// TIA Portal V20 export
DATA_BLOCK "Config"   // DB7
{ DB_Accessible_From_OPC_UA := 'FALSE' }
AUTHOR : ERsystem_FA2_DH. Kim
// stored: DBAccessibleFromOPCUA false, DBAccessibleFromWebserver false, MemoryReserve 100, Namespace Unit1
   VAR
      unit { S7_SetPoint := 'True'} : "LAF_typeUnitConfiguration";   // Configuration of Unit Parameters
      stateMachine { S7_SetPoint := 'True'} : "LUC_typeStateMachineConfiguration";
      signalStack { S7_SetPoint := 'True'} : "LUC_typeSignalStackConfiguration";
      remoteCtrlOpcUa { S7_SetPoint := 'True'} : "LUC_typeRemoteCtrlConfiguration";
      stateModeManager { ExternalAccessible := 'False'; ExternalVisible := 'False'; ExternalWritable := 'False'} : "LPMLV2022_typeConfiguration";   // Do not change. Can be configured through stateMachineConfiguration
      cmPowerMeter_PAC3220 { S7_SetPoint := 'True'} : "LER_typePAC3220Configuration";
      cmHandyQRreadDM8700 { S7_SetPoint := 'True'} : "LER_typeDM8700Configuration";
      cmFFU_LIU117 { S7_SetPoint := 'True'} : "LER_typeLIU117Configuration";
      sleep { S7_SetPoint := 'True'} : "LER_typeSleepModeParameter";
      BA010 : "LER_typeCommunicationConfiguration";
      BA015 : "LER_typeCommunicationConfiguration";
      BA060 : "LER_typeCommunicationConfiguration";
      BA030 : "LER_typeCommunicationConfiguration";
   END_VAR
BEGIN
   unit.referenceDesignator.parent := WSTRING#'';
   unit.referenceDesignator.relative := WSTRING#'STACK#1';
   unit.referenceDesignator.combined := WSTRING#'STACK#1';
   stateMachine.enableModes.production := TRUE;
   stateMachine.enableModes.maintenance := TRUE;
   stateMachine.enableModes.manual := TRUE;
   stateMachine.enableModes.userMode01 := TRUE;   // Enable unit mode NoMode
   stateMachine.enableModes.userMode02 := TRUE;   // Enable unit mode Sleep
   stateMachine.enableModes.userMode03 := TRUE;   // Enable unit mode DeepSleep
   stateMachine.enableModes.userMode04 := FALSE;
   stateMachine.enableModes.userMode05 := FALSE;
   stateMachine.enableModes.userMode06 := FALSE;
   stateMachine.enableModes.userMode07 := FALSE;
   stateMachine.enableModes.userMode08 := FALSE;
   stateMachine.enableModes.userMode09 := FALSE;
   stateMachine.enableModes.userMode10 := FALSE;
   stateMachine.enableModes.userMode11 := FALSE;
   stateMachine.enableModes.userMode12 := FALSE;
   stateMachine.enableModes.userMode13 := FALSE;
   stateMachine.enableStates[0..16].clearing := TRUE;
   stateMachine.enableStates[0..2].starting := TRUE;
   stateMachine.enableStates[3].starting := FALSE;
   stateMachine.enableStates[4..16].starting := TRUE;
   stateMachine.enableStates[0..1].suspended := TRUE;
   stateMachine.enableStates[2..3].suspended := FALSE;
   stateMachine.enableStates[4..16].suspended := TRUE;
   stateMachine.enableStates[0..16].stopping := TRUE;
   stateMachine.enableStates[0..16].aborting := TRUE;
   stateMachine.enableStates[0..2].holding := TRUE;
   stateMachine.enableStates[3].holding := FALSE;
   stateMachine.enableStates[4..16].holding := TRUE;
   stateMachine.enableStates[0..2].held := TRUE;
   stateMachine.enableStates[3].held := FALSE;
   stateMachine.enableStates[4..16].held := TRUE;
   stateMachine.enableStates[0..2].unholding := TRUE;
   stateMachine.enableStates[3].unholding := FALSE;
   stateMachine.enableStates[4..16].unholding := TRUE;
   stateMachine.enableStates[0..1].suspending := TRUE;
   stateMachine.enableStates[2..3].suspending := FALSE;
   stateMachine.enableStates[4..16].suspending := TRUE;
   stateMachine.enableStates[0..1].unsuspending := TRUE;
   stateMachine.enableStates[2..3].unsuspending := FALSE;
   stateMachine.enableStates[4..16].unsuspending := TRUE;
   stateMachine.enableStates[0..16].resetting := TRUE;
   stateMachine.enableStates[0..1].completing := TRUE;
   stateMachine.enableStates[2..3].completing := FALSE;
   stateMachine.enableStates[4..16].completing := TRUE;
   stateMachine.enableStates[0..1].completed := TRUE;
   stateMachine.enableStates[2..3].completed := FALSE;
   stateMachine.enableStates[4..16].completed := TRUE;
   stateMachine.enableModeTransitions[0..16].clearing := FALSE;
   stateMachine.enableModeTransitions[0..16].stopped := TRUE;
   stateMachine.enableModeTransitions[0..16].starting := FALSE;
   stateMachine.enableModeTransitions[0..16].idle := TRUE;
   stateMachine.enableModeTransitions[0..16].suspended := FALSE;
   stateMachine.enableModeTransitions[0..16].execute := FALSE;
   stateMachine.enableModeTransitions[0..16].stopping := FALSE;
   stateMachine.enableModeTransitions[0..16].aborting := FALSE;
   stateMachine.enableModeTransitions[0..16].aborted := TRUE;
   stateMachine.enableModeTransitions[0..16].holding := FALSE;
   stateMachine.enableModeTransitions[0..16].held := FALSE;
   stateMachine.enableModeTransitions[0..16].unholding := FALSE;
   stateMachine.enableModeTransitions[0..16].suspending := FALSE;
   stateMachine.enableModeTransitions[0..16].unsuspending := FALSE;
   stateMachine.enableModeTransitions[0..16].resetting := FALSE;
   stateMachine.enableModeTransitions[0..16].completing := FALSE;
   stateMachine.enableModeTransitions[0..16].completed := FALSE;
   stateMachine.enableHoldCommand.idle := FALSE;
   stateMachine.enableHoldCommand.starting := FALSE;
   stateMachine.enableHoldCommand.suspended := FALSE;
   stateMachine.enableHoldCommand.execute := TRUE;
   stateMachine.enableHoldCommand.unholding := FALSE;
   stateMachine.enableHoldCommand.suspending := FALSE;
   stateMachine.enableHoldCommand.unsuspending := FALSE;
   stateMachine.enableHoldCommand.completing := FALSE;
   stateMachine.enableHoldCommand.completed := FALSE;
   stateMachine.enableCompleteCommand.suspended := TRUE;
   stateMachine.enableCompleteCommand.execute := TRUE;
   stateMachine.enableCompleteCommand.held := TRUE;
   signalStack.undefined.static.red := FALSE;
   signalStack.undefined.static.yellow := FALSE;
   signalStack.undefined.static.blue := FALSE;
   signalStack.undefined.static.green := FALSE;
   signalStack.undefined.static.horn := FALSE;
   signalStack.undefined.static.white := FALSE;
   signalStack.undefined.static.user1 := FALSE;
   signalStack.undefined.static.user2 := FALSE;
   signalStack.undefined.flashing.red := TRUE;
   signalStack.undefined.flashing.yellow := FALSE;
   signalStack.undefined.flashing.blue := FALSE;
   signalStack.undefined.flashing.green := FALSE;
   signalStack.undefined.flashing.horn := FALSE;
   signalStack.undefined.flashing.white := FALSE;
   signalStack.undefined.flashing.user1 := FALSE;
   signalStack.undefined.flashing.user2 := FALSE;
   signalStack.clearing.static.red := FALSE;
   signalStack.clearing.static.yellow := FALSE;
   signalStack.clearing.static.blue := FALSE;
   signalStack.clearing.static.green := FALSE;
   signalStack.clearing.static.horn := FALSE;
   signalStack.clearing.static.white := FALSE;
   signalStack.clearing.static.user1 := FALSE;
   signalStack.clearing.static.user2 := FALSE;
   signalStack.clearing.flashing.red := TRUE;
   signalStack.clearing.flashing.yellow := FALSE;
   signalStack.clearing.flashing.blue := FALSE;
   signalStack.clearing.flashing.green := FALSE;
   signalStack.clearing.flashing.horn := FALSE;
   signalStack.clearing.flashing.white := FALSE;
   signalStack.clearing.flashing.user1 := FALSE;
   signalStack.clearing.flashing.user2 := FALSE;
   signalStack.stopped.static.red := TRUE;
   signalStack.stopped.static.yellow := FALSE;
   signalStack.stopped.static.blue := FALSE;
   signalStack.stopped.static.green := FALSE;
   signalStack.stopped.static.horn := FALSE;
   signalStack.stopped.static.white := FALSE;
   signalStack.stopped.static.user1 := FALSE;
   signalStack.stopped.static.user2 := FALSE;
   signalStack.stopped.flashing.red := FALSE;
   signalStack.stopped.flashing.yellow := FALSE;
   signalStack.stopped.flashing.blue := FALSE;
   signalStack.stopped.flashing.green := FALSE;
   signalStack.stopped.flashing.horn := FALSE;
   signalStack.stopped.flashing.white := FALSE;
   signalStack.stopped.flashing.user1 := FALSE;
   signalStack.stopped.flashing.user2 := FALSE;
   signalStack.starting.static.red := FALSE;
   signalStack.starting.static.yellow := FALSE;
   signalStack.starting.static.blue := FALSE;
   signalStack.starting.static.green := TRUE;
   signalStack.starting.static.horn := FALSE;
   signalStack.starting.static.white := FALSE;
   signalStack.starting.static.user1 := FALSE;
   signalStack.starting.static.user2 := FALSE;
   signalStack.starting.flashing.red := FALSE;
   signalStack.starting.flashing.yellow := FALSE;
   signalStack.starting.flashing.blue := FALSE;
   signalStack.starting.flashing.green := FALSE;
   signalStack.starting.flashing.horn := FALSE;
   signalStack.starting.flashing.white := FALSE;
   signalStack.starting.flashing.user1 := FALSE;
   signalStack.starting.flashing.user2 := FALSE;
   signalStack.idle.static.red := FALSE;
   signalStack.idle.static.yellow := FALSE;
   signalStack.idle.static.blue := FALSE;
   signalStack.idle.static.green := FALSE;
   signalStack.idle.static.horn := FALSE;
   signalStack.idle.static.white := FALSE;
   signalStack.idle.static.user1 := FALSE;
   signalStack.idle.static.user2 := FALSE;
   signalStack.idle.flashing.red := FALSE;
   signalStack.idle.flashing.yellow := FALSE;
   signalStack.idle.flashing.blue := FALSE;
   signalStack.idle.flashing.green := TRUE;
   signalStack.idle.flashing.horn := FALSE;
   signalStack.idle.flashing.white := FALSE;
   signalStack.idle.flashing.user1 := FALSE;
   signalStack.idle.flashing.user2 := FALSE;
   signalStack.suspended.static.red := FALSE;
   signalStack.suspended.static.yellow := TRUE;
   signalStack.suspended.static.blue := FALSE;
   signalStack.suspended.static.green := FALSE;
   signalStack.suspended.static.horn := FALSE;
   signalStack.suspended.static.white := FALSE;
   signalStack.suspended.static.user1 := FALSE;
   signalStack.suspended.static.user2 := FALSE;
   signalStack.suspended.flashing.red := FALSE;
   signalStack.suspended.flashing.yellow := FALSE;
   signalStack.suspended.flashing.blue := FALSE;
   signalStack.suspended.flashing.green := FALSE;
   signalStack.suspended.flashing.horn := FALSE;
   signalStack.suspended.flashing.white := FALSE;
   signalStack.suspended.flashing.user1 := FALSE;
   signalStack.suspended.flashing.user2 := FALSE;
   signalStack.execute.static.red := FALSE;
   signalStack.execute.static.yellow := FALSE;
   signalStack.execute.static.blue := FALSE;
   signalStack.execute.static.green := TRUE;
   signalStack.execute.static.horn := FALSE;
   signalStack.execute.static.white := FALSE;
   signalStack.execute.static.user1 := FALSE;
   signalStack.execute.static.user2 := FALSE;
   signalStack.execute.flashing.red := FALSE;
   signalStack.execute.flashing.yellow := FALSE;
   signalStack.execute.flashing.blue := FALSE;
   signalStack.execute.flashing.green := FALSE;
   signalStack.execute.flashing.horn := FALSE;
   signalStack.execute.flashing.white := FALSE;
   signalStack.execute.flashing.user1 := FALSE;
   signalStack.execute.flashing.user2 := FALSE;
   signalStack.stopping.static.red := TRUE;
   signalStack.stopping.static.yellow := FALSE;
   signalStack.stopping.static.blue := FALSE;
   signalStack.stopping.static.green := FALSE;
   signalStack.stopping.static.horn := FALSE;
   signalStack.stopping.static.white := FALSE;
   signalStack.stopping.static.user1 := FALSE;
   signalStack.stopping.static.user2 := FALSE;
   signalStack.stopping.flashing.red := FALSE;
   signalStack.stopping.flashing.yellow := FALSE;
   signalStack.stopping.flashing.blue := FALSE;
   signalStack.stopping.flashing.green := FALSE;
   signalStack.stopping.flashing.horn := FALSE;
   signalStack.stopping.flashing.white := FALSE;
   signalStack.stopping.flashing.user1 := FALSE;
   signalStack.stopping.flashing.user2 := FALSE;
   signalStack.aborting.static.red := FALSE;
   signalStack.aborting.static.yellow := FALSE;
   signalStack.aborting.static.blue := FALSE;
   signalStack.aborting.static.green := FALSE;
   signalStack.aborting.static.horn := FALSE;
   signalStack.aborting.static.white := FALSE;
   signalStack.aborting.static.user1 := FALSE;
   signalStack.aborting.static.user2 := FALSE;
   signalStack.aborting.flashing.red := TRUE;
   signalStack.aborting.flashing.yellow := FALSE;
   signalStack.aborting.flashing.blue := FALSE;
   signalStack.aborting.flashing.green := FALSE;
   signalStack.aborting.flashing.horn := FALSE;
   signalStack.aborting.flashing.white := FALSE;
   signalStack.aborting.flashing.user1 := FALSE;
   signalStack.aborting.flashing.user2 := FALSE;
   signalStack.aborted.static.red := FALSE;
   signalStack.aborted.static.yellow := FALSE;
   signalStack.aborted.static.blue := FALSE;
   signalStack.aborted.static.green := FALSE;
   signalStack.aborted.static.horn := FALSE;
   signalStack.aborted.static.white := FALSE;
   signalStack.aborted.static.user1 := FALSE;
   signalStack.aborted.static.user2 := FALSE;
   signalStack.aborted.flashing.red := TRUE;
   signalStack.aborted.flashing.yellow := FALSE;
   signalStack.aborted.flashing.blue := FALSE;
   signalStack.aborted.flashing.green := FALSE;
   signalStack.aborted.flashing.horn := FALSE;
   signalStack.aborted.flashing.white := FALSE;
   signalStack.aborted.flashing.user1 := FALSE;
   signalStack.aborted.flashing.user2 := FALSE;
   signalStack.holding.static.red := FALSE;
   signalStack.holding.static.yellow := FALSE;
   signalStack.holding.static.blue := FALSE;
   signalStack.holding.static.green := FALSE;
   signalStack.holding.static.horn := FALSE;
   signalStack.holding.static.white := FALSE;
   signalStack.holding.static.user1 := FALSE;
   signalStack.holding.static.user2 := FALSE;
   signalStack.holding.flashing.red := FALSE;
   signalStack.holding.flashing.yellow := FALSE;
   signalStack.holding.flashing.blue := TRUE;
   signalStack.holding.flashing.green := FALSE;
   signalStack.holding.flashing.horn := FALSE;
   signalStack.holding.flashing.white := FALSE;
   signalStack.holding.flashing.user1 := FALSE;
   signalStack.holding.flashing.user2 := FALSE;
   signalStack.held.static.red := FALSE;
   signalStack.held.static.yellow := FALSE;
   signalStack.held.static.blue := TRUE;
   signalStack.held.static.green := FALSE;
   signalStack.held.static.horn := FALSE;
   signalStack.held.static.white := FALSE;
   signalStack.held.static.user1 := FALSE;
   signalStack.held.static.user2 := FALSE;
   signalStack.held.flashing.red := FALSE;
   signalStack.held.flashing.yellow := FALSE;
   signalStack.held.flashing.blue := FALSE;
   signalStack.held.flashing.green := FALSE;
   signalStack.held.flashing.horn := FALSE;
   signalStack.held.flashing.white := FALSE;
   signalStack.held.flashing.user1 := FALSE;
   signalStack.held.flashing.user2 := FALSE;
   signalStack.unholding.static.red := FALSE;
   signalStack.unholding.static.yellow := FALSE;
   signalStack.unholding.static.blue := FALSE;
   signalStack.unholding.static.green := TRUE;
   signalStack.unholding.static.horn := FALSE;
   signalStack.unholding.static.white := FALSE;
   signalStack.unholding.static.user1 := FALSE;
   signalStack.unholding.static.user2 := FALSE;
   signalStack.unholding.flashing.red := FALSE;
   signalStack.unholding.flashing.yellow := FALSE;
   signalStack.unholding.flashing.blue := FALSE;
   signalStack.unholding.flashing.green := FALSE;
   signalStack.unholding.flashing.horn := FALSE;
   signalStack.unholding.flashing.white := FALSE;
   signalStack.unholding.flashing.user1 := FALSE;
   signalStack.unholding.flashing.user2 := FALSE;
   signalStack.suspending.static.red := FALSE;
   signalStack.suspending.static.yellow := FALSE;
   signalStack.suspending.static.blue := FALSE;
   signalStack.suspending.static.green := FALSE;
   signalStack.suspending.static.horn := FALSE;
   signalStack.suspending.static.white := FALSE;
   signalStack.suspending.static.user1 := FALSE;
   signalStack.suspending.static.user2 := FALSE;
   signalStack.suspending.flashing.red := FALSE;
   signalStack.suspending.flashing.yellow := TRUE;
   signalStack.suspending.flashing.blue := FALSE;
   signalStack.suspending.flashing.green := FALSE;
   signalStack.suspending.flashing.horn := FALSE;
   signalStack.suspending.flashing.white := FALSE;
   signalStack.suspending.flashing.user1 := FALSE;
   signalStack.suspending.flashing.user2 := FALSE;
   signalStack.unsuspending.static.red := FALSE;
   signalStack.unsuspending.static.yellow := FALSE;
   signalStack.unsuspending.static.blue := FALSE;
   signalStack.unsuspending.static.green := TRUE;
   signalStack.unsuspending.static.horn := FALSE;
   signalStack.unsuspending.static.white := FALSE;
   signalStack.unsuspending.static.user1 := FALSE;
   signalStack.unsuspending.static.user2 := FALSE;
   signalStack.unsuspending.flashing.red := FALSE;
   signalStack.unsuspending.flashing.yellow := FALSE;
   signalStack.unsuspending.flashing.blue := FALSE;
   signalStack.unsuspending.flashing.green := FALSE;
   signalStack.unsuspending.flashing.horn := FALSE;
   signalStack.unsuspending.flashing.white := FALSE;
   signalStack.unsuspending.flashing.user1 := FALSE;
   signalStack.unsuspending.flashing.user2 := FALSE;
   signalStack.resetting.static.red := TRUE;
   signalStack.resetting.static.yellow := FALSE;
   signalStack.resetting.static.blue := FALSE;
   signalStack.resetting.static.green := FALSE;
   signalStack.resetting.static.horn := FALSE;
   signalStack.resetting.static.white := FALSE;
   signalStack.resetting.static.user1 := FALSE;
   signalStack.resetting.static.user2 := FALSE;
   signalStack.resetting.flashing.red := FALSE;
   signalStack.resetting.flashing.yellow := FALSE;
   signalStack.resetting.flashing.blue := FALSE;
   signalStack.resetting.flashing.green := FALSE;
   signalStack.resetting.flashing.horn := FALSE;
   signalStack.resetting.flashing.white := FALSE;
   signalStack.resetting.flashing.user1 := FALSE;
   signalStack.resetting.flashing.user2 := FALSE;
   signalStack.completing.static.red := FALSE;
   signalStack.completing.static.yellow := FALSE;
   signalStack.completing.static.blue := FALSE;
   signalStack.completing.static.green := TRUE;
   signalStack.completing.static.horn := FALSE;
   signalStack.completing.static.white := FALSE;
   signalStack.completing.static.user1 := FALSE;
   signalStack.completing.static.user2 := FALSE;
   signalStack.completing.flashing.red := FALSE;
   signalStack.completing.flashing.yellow := FALSE;
   signalStack.completing.flashing.blue := FALSE;
   signalStack.completing.flashing.green := FALSE;
   signalStack.completing.flashing.horn := FALSE;
   signalStack.completing.flashing.white := FALSE;
   signalStack.completing.flashing.user1 := FALSE;
   signalStack.completing.flashing.user2 := FALSE;
   signalStack.completed.static.red := TRUE;
   signalStack.completed.static.yellow := FALSE;
   signalStack.completed.static.blue := FALSE;
   signalStack.completed.static.green := FALSE;
   signalStack.completed.static.horn := FALSE;
   signalStack.completed.static.white := FALSE;
   signalStack.completed.static.user1 := FALSE;
   signalStack.completed.static.user2 := FALSE;
   signalStack.completed.flashing.red := FALSE;
   signalStack.completed.flashing.yellow := FALSE;
   signalStack.completed.flashing.blue := FALSE;
   signalStack.completed.flashing.green := FALSE;
   signalStack.completed.flashing.horn := FALSE;
   signalStack.completed.flashing.white := FALSE;
   signalStack.completed.flashing.user1 := FALSE;
   signalStack.completed.flashing.user2 := FALSE;
   remoteCtrlOpcUa.enableMethods.reset := TRUE;
   remoteCtrlOpcUa.enableMethods.start := TRUE;
   remoteCtrlOpcUa.enableMethods.stop := TRUE;
   remoteCtrlOpcUa.enableMethods.hold := TRUE;
   remoteCtrlOpcUa.enableMethods.unhold := TRUE;
   remoteCtrlOpcUa.enableMethods.suspend := TRUE;
   remoteCtrlOpcUa.enableMethods.unsuspend := TRUE;
   remoteCtrlOpcUa.enableMethods.abort := TRUE;
   remoteCtrlOpcUa.enableMethods.clear := TRUE;
   remoteCtrlOpcUa.enableMethods.complete := TRUE;
   remoteCtrlOpcUa.enableMethods.stateComplete := TRUE;
   remoteCtrlOpcUa.enableMethods.requestUnitMode := TRUE;
   remoteCtrlOpcUa.enableMethods.requestUnitState := TRUE;
   stateModeManager.EnabledModesCfg := 16#0000_007F;
   stateModeManager.DisabledStatesCfg[0..1] := 16#0000_0000;
   stateModeManager.DisabledStatesCfg[2] := 16#0003_6020;
   stateModeManager.DisabledStatesCfg[3] := 16#0003_7C28;
   stateModeManager.DisabledStatesCfg[4..16] := 16#0000_0000;
   stateModeManager.ModeTransitionCfg[0..16] := 16#0000_0214;
   stateModeManager.holdCmdCfg := 16#0000_0040;
   stateModeManager.completeCmdCfg := 16#0000_0860;
   BA010.disableAlarms := FALSE;
   BA010.SEND.connectionId := 16#0112;
   BA010.SEND.rid := 16#0000_0021;
   BA010.SEND.len := 16#0000;
   BA010.RCV.connectionId := 16#0112;
   BA010.RCV.rid := 16#0000_0022;
   BA015.disableAlarms := FALSE;
   BA015.SEND.connectionId := 16#0117;
   BA015.SEND.rid := 16#0000_0023;
   BA015.SEND.len := 16#0000;
   BA015.RCV.connectionId := 16#0117;
   BA015.RCV.rid := 16#0000_0024;
   BA060.disableAlarms := FALSE;
   BA060.SEND.connectionId := 16#0162;
   BA060.SEND.rid := 16#0000_0025;
   BA060.SEND.len := 16#0000;
   BA060.RCV.connectionId := 16#0162;
   BA060.RCV.rid := 16#0000_0026;
   BA030.disableAlarms := FALSE;
   BA030.SEND.connectionId := 16#0142;
   BA030.SEND.rid := 16#0000_0018;
   BA030.SEND.len := 16#0000;
   BA030.RCV.connectionId := 16#0142;
   BA030.RCV.rid := 16#0000_0017;
END_DATA_BLOCK
